// TIA Portal V19 export
VAR_GLOBAL   // PLC tag table "D07"
   D07_Lp_EntryReq_LB123 AT %Q107.6 : Bool;   // 194SH1
   D07_Lp_SafetyReset_LB123 AT %Q107.7 : Bool;   // 194SH2
   D07_Pb_EntryReq_LB123 AT %I104.4 : Bool;   // 194SH1
   D07_Pb_SafetyReset_LB123 AT %I104.5 : Bool;   // 194SH2
   D07_Unlock AT %Q107.5 : Bool;   // 19402 Comando_Elettroserratura
   D07_LockEnable AT %I104.2 : Bool;   // 19401 Cancello chiuso
   D07_Cancello_Bloccato AT %I104.3 : Bool;   // 19403
   D07_Ls AT %I1027.1 : Bool;   // 103DI1 - 194A1
END_VAR
